// TwinCAT 3 PLC project PLC1
// ProgramVersion: 3.1.4026.15
// libraries:
//   Tc2_Standard, * (Beckhoff Automation GmbH)
//   Tc2_System, * (Beckhoff Automation GmbH)
// project tree:
//   / PlcTask.TcTTO (not stored)
//   POUs/ MAIN.TcPOU
// real-time tasks:
//   TASK PlcTask: cycle T#10ms, priority 20, ADS port 350
// motion (NC):
//   TASK NC-Task 1 SAF: cycle T#2ms, priority 4, ADS port 501
//   TASK NC-Task 1 SVB: cycle T#10ms, priority 8, ADS port 511
//   AXIS Axis 1 (id 1)
//     OtherSettings: AllowMotionCmdToSlave=true
//     encoder EncType=19
//       EncPara: MaxCount=#xffffffff
//     drive DrvType=16
//       DrvPara: MaxCount=#xffffffff, DriveControlDWord=#x00020000
//         Analog: TorqueSetpointScale=10, ScaleFactorActTorque=0.1
//         TimeComp: TaskDelayCycles=1
//     controller CtrType=1
//       CtrPara: PriorControlFactor=1
//         Observer: BandWidth=20
// I/O:
//   DEVICE Device 1 (EtherCAT), AmsNetId 10.200.70.2.2.1
//     Term 1 (EK1200) [EK1200-5000 EtherCAT Power supply (2A E-Bus)]
//       Term 2 (EL1859) [EL1859 8Ch. Dig. Input 24V, 3ms, 8Ch. Dig. Output 24V, 0.5A]
//       Term 3 (EL1859) [EL1859 8Ch. Dig. Input 24V, 3ms, 8Ch. Dig. Output 24V, 0.5A]
//       Term 4 (EL3255) [EL3255 5Ch. potentiometer measurement with sensor supply]
//       Term 5 (EL3214-0090) [EL3214-0090 4Ch. Ana. Input PT100 (RTD), TwinSAFE SC]
//       Term 6 (EL5151) [EL5151 1Ch. Inc. Encoder]
//       Term 7 (EL1918) [EL1918, 8Ch. Safety Input 24V, TwinSAFE]
//         modules: Module 2 (FSLOGIC)
//       Term 8 (EL2912) [EL2912, 2Ch. Safety Output 24V, 2A, TwinSAFE]
//         modules: Module 1 (FSOE), Module 2 (FSOUT), Module 3 (DEVICEIO), Module 4 (FSLOGIC)
//       Term 9 (EL9110) [EL9110 Power Supplier with LED (24V, Diagnostics)]
//       Term 10 (EL7201-9014) [EL7201-9014 1Ch. MDP742 Servo motor output stage with OCT (50V, 2.8A RMS) and STO input]
//       Term 11 (EK1122) [EK1122 2 port EtherCAT junction]
//       Term 12 (EL9011) [EL9011 End Terminal]
//   DEVICE Device 2 (EtherCAT Automation Protocol), AmsNetId 10.200.70.2.3.1
//     publisher-1
//     subscriber-1
//     publisher-2
//     subscriber-2
// variable links:
//   Device 1 (EtherCAT) <-> Device 2 (EtherCAT Automation Protocol)/publisher-1
//     Term 1 (EK1200)/Term 7 (EL1918)/ConnectionInputs/Message_5 TxPDO <-> safe-data-out/Outputs/VarData
//   Device 1 (EtherCAT) <-> Device 2 (EtherCAT Automation Protocol)/publisher-2
//     Term 1 (EK1200)/Term 7 (EL1918)/ConnectionInputs/Message_6 TxPDO <-> safe-data-out/Outputs/VarData
//   Device 1 (EtherCAT) <-> Device 2 (EtherCAT Automation Protocol)/subscriber-1
//     Term 1 (EK1200)/Term 7 (EL1918)/ConnectionOutputs/Message_5 RxPDO <-> safe-data-in/Inputs/VarData
//   Device 1 (EtherCAT) <-> Device 2 (EtherCAT Automation Protocol)/subscriber-2
//     Term 1 (EK1200)/Term 7 (EL1918)/ConnectionOutputs/Message_6 RxPDO <-> safe-data-in/Inputs/VarData
//   NC-Task 1 SAF/Axes/Axis 1 <-> Device 1 (EtherCAT)/Term 1 (EK1200)/Term 10 (EL7201-9014)
//     Drive/Inputs/In/nDcOutputTime <-> InfoData/DcOutputShift
//     Drive/Inputs/In/nState1 <-> DRV Statusword/Statusword
//     Drive/Inputs/In/nState2 <-> DRV Statusword/Statusword @bit 8
//     Drive/Inputs/In/nState4 @bit 1 <-> WcState/InputToggle
//     Drive/Inputs/In/nState4 <-> WcState/WcState
//     Drive/Outputs/Out/nCtrl1 <-> DRV Controlword/Controlword
//     Drive/Outputs/Out/nCtrl2 <-> DRV Controlword/Controlword @bit 8
//     Drive/Outputs/Out/nDataOut2 <-> DRV Target velocity/Target velocity
//     Enc/Inputs/In/nDataIn1 <-> FB Position/Position
//     Enc/Inputs/In/nDcInputTime <-> InfoData/DcInputShift
//     Enc/Inputs/In/nState4 @bit 1 <-> WcState/InputToggle
//     Enc/Inputs/In/nState4 <-> WcState/WcState
//   PLC1/PLC1 Instance <-> Device 1 (EtherCAT)/Term 1 (EK1200)/Term 7 (EL1918)
//     PlcTask Outputs/MAIN.safe_err_ack <-> StandardOutputs/Standard In Var 1
//     PlcTask Outputs/MAIN.safe_run <-> StandardOutputs/Standard In Var 2
//   PLC1/PLC1 Instance <-> Device 2 (EtherCAT Automation Protocol)/publisher-1
//     PlcTask Outputs/MAIN.com_check_pub <-> com-check-out/Outputs/VarData
//   PLC1/PLC1 Instance <-> Device 2 (EtherCAT Automation Protocol)/subscriber-1
//     PlcTask Inputs/MAIN.com_check_sub <-> com-check-in/Inputs/VarData

// ---- POUs/MAIN.TcPOU
PROGRAM MAIN
VAR
	safe_err_ack AT %Q* : BOOL;
	safe_run AT %Q* : BOOL;
	safe_reset AT %Q* : BOOL;
	
	com_check_pub AT %Q* : BOOL;
	com_check_sub AT %I* : BOOL;
	
END_VAR

END_PROGRAM
